FUNCTION F_LaserSetpoints : ST_LaserSetpoints
VAR_INPUT
END_VAR
VAR
	stSetpoints : ST_LaserSetpoints := (
		nMinVoltage := 2,
		nMinNominalVoltage := 4
	);
END_VAR

F_LaserSetpoints := stSetpoints;

END_FUNCTION

(* stored: Version 1.1.0.1, ProductVersion 3.1.4020.14
   POU F_LaserSetpoints: Id {a52d574d-6658-40ce-ae47-23dd58ff0f5e}, SpecialFunc None *)
